KUKA KRL program: start_weld_respot.src

&ACCESS RVO2
&REL 149
&COMMENT start_weld_RESPOT
&PARAM DISKPATH = KRC:\R1\Program\SubRotinas
DEF start_weld_RESPOT( )
;
;FOLD OUT 3334 'R2 solda respot Ok' State=FALSE ;%{PE}%R 8.2.20,%MKUKATPBASIS,%COUT,%VOUTX,%P 2:3334, 3:R2 solda respot Ok, 5:FALSE, 6:
$OUT[3334]=FALSE
;ENDFOLD
;
END
